// 隐含生成代码：不要编辑
FUNCTION CheckLRangeSigned : LINT
VAR_INPUT
	value, lower, upper: LINT;
END_VAR

// 隐含生成代码：这里只是对代码实现的建议
{noflow}
IF (value < lower) THEN
	CheckLRangeSigned := lower;
ELSIF(value > upper) THEN
	CheckLRangeSigned := upper;
ELSE
	CheckLRangeSigned := value;
END_IF

{flow}

END_FUNCTION

(* stored: Version 1.1.0.1, ProductVersion 3.1.4024.9
   POU CheckLRangeSigned: Id {faf15c6d-3606-4ef1-a185-c772e31d1e84}, SpecialFunc CheckLRangeSigned *)
